PROGRAM P_MQTT_Agent
VAR
	fbIoTManager			:	FB_IotMqttClient;
    fbMessageQueue 			: 	FB_IotMqttMessageQueue;
    fbMessage      			: 	FB_IotMqttMessage;
    fbGetSystemTime         : GETSYSTEMTIME;
    fileTime        		: T_FILETIME;
	
	bTopicsSubscribed		:	BOOL;
	bConfigured				:	BOOL;
	sBuffer					:	STRING;
END_VAR

IF NOT bConfigured THEN 
	bConfigured := TRUE;
	
	fbIoTManager.sHostName  := GVL_MQTT_Conf.sServerIp;
	fbIoTManager.nHostPort	:= GVL_MQTT_Conf.sServerPort;
	fbIoTManager.sTopicPrefix := CONCAT(STR1 := GVL_MQTT_Conf.sMainTopic,str2 := 
												concat(str1 := '/',STR2 := GVL_MQTT_Conf.sDevice));
	fbIoTManager.ipMessageQueue	:=	fbMessageQueue;
ELSE
	fbIoTManager.Execute(bConnect := TRUE);
END_IF


IF fbIoTManager.bConnected AND NOT bTopicsSubscribed THEN 
	M_SubscribeToTopics();
END_IF

IF fbMessageQueue.nQueuedMessages <> 0 THEN 
	fbMessageQueue.Dequeue(fbMessage := fbMessage);
	
	IF fbMessage.CompareTopic(sTopic := GVL_MQTT_Conf.sFullBatTopic) THEN
		fbMessage.GetPayload(pPayload := ADR(sBuffer),
							nPayloadSize := fbMessage.nPayloadSize,
							bSetNullTermination := FALSE);
		GVL_ShellyRecentValues.iBatteryLevel := STRING_TO_INT(sBuffer);
	ELSIF fbMessage.CompareTopic(sTopic := GVL_MQTT_Conf.sFullHumTopic) THEN
		fbMessage.GetPayload(pPayload := ADR(sBuffer),
							nPayloadSize := fbMessage.nPayloadSize,
							bSetNullTermination := FALSE);
		GVL_ShellyRecentValues.rHumidity := STRING_TO_REAL(sBuffer);
	ELSIF fbMessage.CompareTopic(sTopic := GVL_MQTT_Conf.sFullTempTopic) THEN
		fbMessage.GetPayload(pPayload := ADR(sBuffer),
							nPayloadSize := fbMessage.nPayloadSize,
							bSetNullTermination := FALSE);
		GVL_ShellyRecentValues.rTemperature := STRING_TO_REAL(sBuffer);
	END_IF
	
	IF fbMessageQueue.nQueuedMessages  = 0 THEN 
		fbGetSystemTime(timeLoDW=>fileTime.dwLowDateTime, timeHiDW=>fileTime.dwHighDateTime );
		GVL_MQTT_Conf.sTimeStamp :=SYSTEMTIME_TO_STRING( FILETIME_TO_SYSTEMTIME( fileTime ) );
		GVL_MQTT_Common.bNewDataJustCame := TRUE;
	END_IF
	
END_IF








IF GVL_MQTT_Common.bRestartServer THEN
	M_NewConf();
	GVL_MQTT_Common.bRestartServer := FALSE;
	M_UnsubscribeToTopics();
END_IF
GVL_MQTT_Conf.bConnected	:=	fbIoTManager.bConnected;
GVL_MQTT_Conf.bErr			:=	fbIoTManager.bError;
GVL_MQTT_Conf.hrErrCode		:=	fbIoTManager.hrErrorCode;

METHOD M_NewConf : BOOL
VAR_INPUT
END_VAR
bConfigured := FALSE;
fbIoTManager.Execute(bConnect := false);
END_METHOD

METHOD M_SubscribeToTopics : BOOL
VAR_INPUT
END_VAR
IF 		fbIoTManager.Subscribe(sTopic := GVL_MQTT_Conf.sHumTopic,eQoS := TcIotMqttQos.ExactlyOnceDelivery)AND
	fbIoTManager.Subscribe(sTopic := GVL_MQTT_Conf.sTempTopic,eQoS := TcIotMqttQos.ExactlyOnceDelivery)AND
	fbIoTManager.Subscribe(sTopic := GVL_MQTT_Conf.sBatTopic,eQoS := TcIotMqttQos.ExactlyOnceDelivery) THEN
	M_SubscribeToTopics := FALSE;
	bTopicsSubscribed := TRUE;
	GVL_MQTT_Conf.sFullBatTopic := CONCAT(STR1 := fbIoTManager.sTopicPrefix,STR2:= GVL_MQTT_Conf.sBatTopic);
	GVL_MQTT_Conf.sFullHumTopic := CONCAT(STR1 := fbIoTManager.sTopicPrefix,STR2:= GVL_MQTT_Conf.sHumTopic);
	GVL_MQTT_Conf.sFullTempTopic := CONCAT(STR1 := fbIoTManager.sTopicPrefix,STR2:= GVL_MQTT_Conf.sTempTopic);
ELSE
	M_SubscribeToTopics := TRUE;
END_IF
END_METHOD

METHOD M_UnsubscribeToTopics : BOOL
VAR_INPUT
END_VAR
IF 	fbIoTManager.Unsubscribe(sTopic := GVL_MQTT_Conf.sHumTopic)AND
	fbIoTManager.Unsubscribe(sTopic := GVL_MQTT_Conf.sTempTopic)AND
	fbIoTManager.Unsubscribe(sTopic := GVL_MQTT_Conf.sBatTopic) THEN
	M_UnsubscribeToTopics := FALSE;
	bTopicsSubscribed := FALSE;
ELSE
	M_UnsubscribeToTopics := TRUE;
END_IF
END_METHOD

END_PROGRAM

(* stored: Version 1.1.0.1, ProductVersion 3.1.4024.9
   POU P_MQTT_Agent: Id {1d7d88b9-4e82-49ca-85cd-baf5c6d87290}, SpecialFunc None
   Method M_NewConf: Id {5903465c-c96d-4e86-8700-c780b8d640bd}
   Method M_SubscribeToTopics: Id {0d7ca85b-4eb3-4834-99a9-4c6698a036c6}
   Method M_UnsubscribeToTopics: Id {efaf8946-48e6-4047-ae3d-8a410e04841c} *)
